PROGRAM P_Demo_STRING_TO_WSTRING2
VAR
    sLocal   : STRING(1024) := 'Long log line...'; // 工业语义：长 STRING
    wsOut    : WSTRING(1024); // 转换后 WSTRING
    bOk      : BOOL; // 完整转换
    bConvert : BOOL; // 在线触发
END_VAR

// =============================================================================
// 场景：HMI 模块用 WSTRING 显示多语言字符串；从配置文件读出的 STRING 配置项需要转 WSTRING 才能显示。
// 价值：`Tc2_Standard` 的 255 限制；本函数无限制。
// 验证步骤：
//   1. 引用 Tc2_Utilities
//   2. 编译 + 登录 + 运行
//   3. 在线写触发位 TRUE，monitor 输出变量
// =============================================================================
IF bConvert THEN
    bOk := STRING_TO_WSTRING2(pDstWSTRING := ADR(wsOut),
                              pSrcSTRING  := ADR(sLocal),
                              nDstSize    := SIZEOF(wsOut));
    bConvert := FALSE;
END_IF;

END_PROGRAM

(* stored: Version 1.1.0.1, ProductVersion 3.1.4024.5
   POU P_Demo_STRING_TO_WSTRING2: Id {59cf749a-3d9d-5017-8fe0-4e29189a1519}, SpecialFunc None *)
